TYPE ST_SEC_ZXX7_ActiveExceptions :
STRUCT
	DeviceWarning		: BOOL;
	DeviceError			: BOOL;
	ManufacturerWarning	: BOOL;
	ManufacturerError	: BOOL;
END_STRUCT
END_TYPE

(* stored: Version 1.1.0.1, ProductVersion 3.1.4024.15
   DUT ST_SEC_ZXX7_ActiveExceptions: Id {849d8a37-1509-02c9-190d-d4fc8bfe6ac8} *)
